SUBAPPLICATION Softkey_IXA_TO_logiBUS_QXA_BG (* Konvertierung Softkey IXA zu logiBUS QXA und Background *)
  (* Standard: 61499-2; Description: Copyright (c) 2023 Meisterschulen am Ostbahnhof This program and the accompanying materials are made available under the terms of the Eclipse Public License 2.0 which is available at https://www.eclipse.org/legal/epl-2.0/ SPDX-License-Identifier: EPL-2.0 *)
  (* Version 1.1, 2026-07-20, Franz Höpfinger, Meisterschulen am Ostbahnhof, Background *)
  (* Version 1.0, 2026-01-15, Franz Höpfinger, Meisterschulen am Ostbahnhof, initial API and implementation and/or initial documentation *)
  PACKAGE MyLib::sys;
  IMPORT isobus::UT::Q::const::IDs::ID_NULL;
  IMPORT logiBUS::io::DQ::logiBUS_DO;
  IMPORT logiBUS::io::DQ::logiBUS_DO_S;
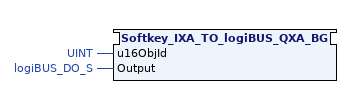
  VAR_INPUT
    u16ObjId : UINT := ID_NULL; (* Object ID *)
    Output : logiBUS::io::DQ::logiBUS_DO_S := logiBUS_DO::Invalid; (* Identify the Output Output_Q1..Q8 *)
  END_VAR
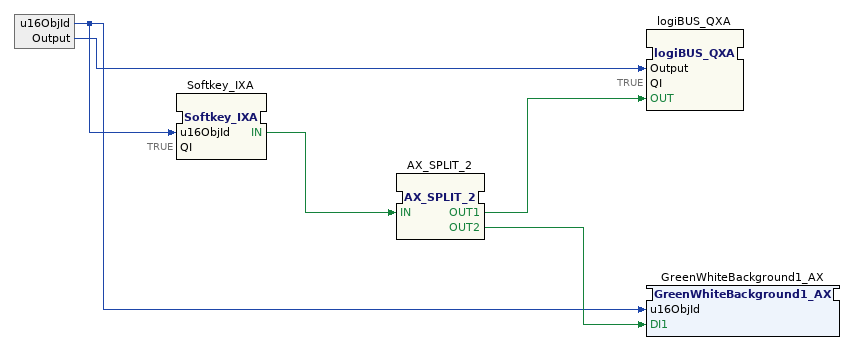
  FBS
    logiBUS_QXA : logiBUS::io::DQ::logiBUS_QXA(QI := TRUE);
    Softkey_IXA : isobus::UT::io::Softkey::Softkey_IXA(QI := TRUE);
    AX_SPLIT_2 : adapter::events::unidirectional::AX_SPLIT_2;
  END_FBS
  SUBAPPS
    GreenWhiteBackground1_AX : MyLib::sys::GreenWhiteBackground1_AX;
  END_SUBAPPS
  DATA_CONNECTIONS
    u16ObjId TO Softkey_IXA.u16ObjId;
    Output TO logiBUS_QXA.Output;
    u16ObjId TO GreenWhiteBackground1_AX.u16ObjId;
  END_CONNECTIONS
  ADAPTER_CONNECTIONS
    Softkey_IXA.IN TO AX_SPLIT_2.IN;
    AX_SPLIT_2.OUT1 TO logiBUS_QXA.OUT;
    AX_SPLIT_2.OUT2 TO GreenWhiteBackground1_AX.DI1;
  END_CONNECTIONS
END_SUBAPPLICATION
